{attribute addProperty BoxType "EL3611-1030-0016"}
{attribute addProperty Id "StatusAT %I*Status_C6F82E6F1621ValueAT %I*DINT32417"}
{attribute addProperty CRC "3201558924"}
{attribute addProperty SizeInBites "48"}
{attribute addProperty SizeInBytes "6"}
TYPE AI_Inputs_BED3E98C :
STRUCT
	{attribute addProperty Name "Status"}
	Status AT %I* : Status_C6F82E6F;
	{attribute addProperty Name "Value"}
	Value AT %I* : DINT;
END_STRUCT
END_TYPE

(* stored: Version 1.2.0.0, ProductVersion 3.1.4024.9
   DUT AI_Inputs_BED3E98C: Id {b788e099-ded0-460c-82ef-2eb2e2b0a11d} *)
